TYPE DTM_Mes1 :	//XFP20240315
STRUCT
	uOther		:ARRAY[0..19] OF UINT;	//信号交互		
	bFuncEN     :ARRAY[0..10] OF BOOL; //功能开关状态
END_STRUCT
END_TYPE

(* stored: Version 1.1.0.1, ProductVersion 3.1.4024.12
   DUT DTM_Mes1: Id {e153ba22-9fa0-4354-b44e-9fc8eaf41d83} *)
